Fanuc KAREL source: kt00706.KL

-- PROVISIONAL review KL for V770-1; original PC SHA256 aa26bd0740d413c9df4a90d2e924d2fa0e5e9e3220cf88d93b85f8ac43bc0de5
-- Incomplete behavior may be omitted. Consult companion uncertainty JSON. Do not deploy.
PROGRAM KT00706
%NOLOCKGROUP
VAR
  I1 : INTEGER
  I2 : INTEGER
  OUT : BOOLEAN
BEGIN
  -- UNRESOLVED_PC offsets 5-16; opcodes 2E,23
  -- UNRESOLVED_PC offsets 21-32; opcodes 2E,23
  -- UNRESOLVED_PC offsets 37-48; opcodes 2E,23
  -- UNRESOLVED_PC offsets 53-64; opcodes 2E,23
  -- UNRESOLVED_PC offsets 69-84; opcodes 22,63,23
  -- UNRESOLVED_PC offsets 89-93; opcodes 7F
END KT00706
